PROGRAM Axis_06_Function_Blocks
VAR
END_VAR

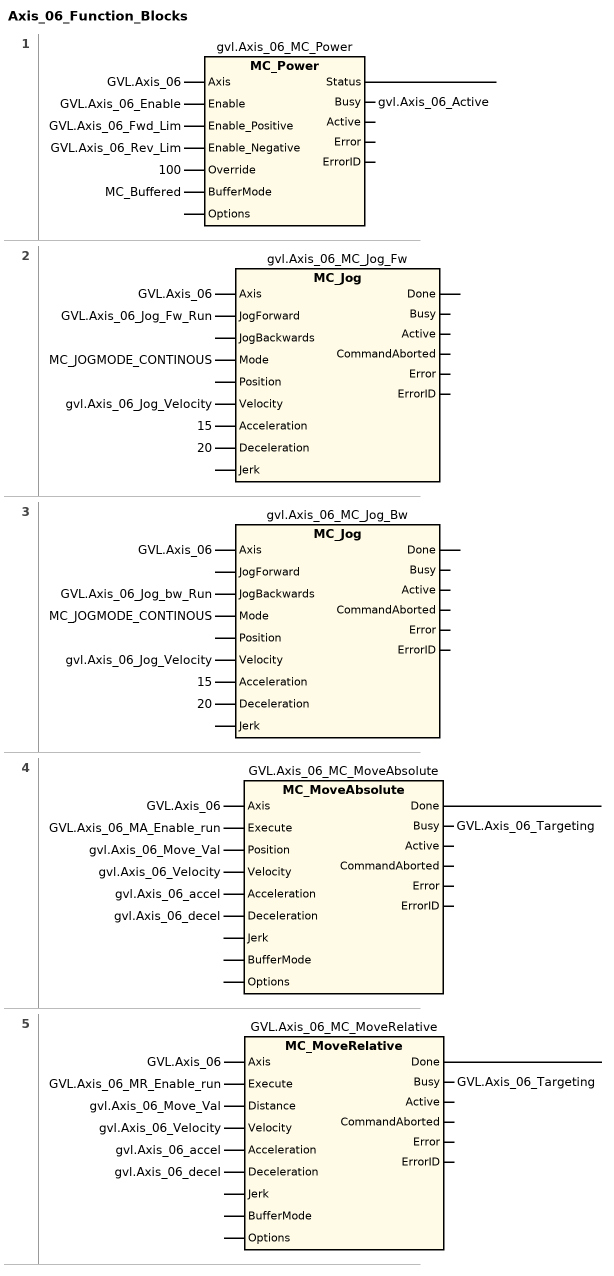
// NETWORK 1
gvl.Axis_06_MC_Power(
    Axis := GVL.Axis_06,
    Enable := GVL.Axis_06_Enable,
    Enable_Positive := GVL.Axis_06_Fwd_Lim,
    Enable_Negative := GVL.Axis_06_Rev_Lim,
    Override := 100,
    BufferMode := MC_Buffered,
    Busy => gvl.Axis_06_Active); // MC_Power

// NETWORK 2
gvl.Axis_06_MC_Jog_Fw(
    Axis := GVL.Axis_06,
    JogForward := GVL.Axis_06_Jog_Fw_Run,
    Mode := MC_JOGMODE_CONTINOUS,
    Velocity := gvl.Axis_06_Jog_Velocity,
    Acceleration := 15,
    Deceleration := 20); // MC_Jog

// NETWORK 3
gvl.Axis_06_MC_Jog_Bw(
    Axis := GVL.Axis_06,
    JogBackwards := GVL.Axis_06_Jog_bw_Run,
    Mode := MC_JOGMODE_CONTINOUS,
    Velocity := gvl.Axis_06_Jog_Velocity,
    Acceleration := 15,
    Deceleration := 20); // MC_Jog

// NETWORK 4
GVL.Axis_06_MC_MoveAbsolute(
    Axis := GVL.Axis_06,
    Execute := GVL.Axis_06_MA_Enable_run,
    Position := gvl.Axis_06_Move_Val,
    Velocity := gvl.Axis_06_Velocity,
    Acceleration := gvl.Axis_06_accel,
    Deceleration := gvl.Axis_06_decel,
    Busy => GVL.Axis_06_Targeting); // MC_MoveAbsolute

// NETWORK 5
GVL.Axis_06_MC_MoveRelative(
    Axis := GVL.Axis_06,
    Execute := GVL.Axis_06_MR_Enable_run,
    Distance := gvl.Axis_06_Move_Val,
    Velocity := gvl.Axis_06_Velocity,
    Acceleration := gvl.Axis_06_accel,
    Deceleration := gvl.Axis_06_decel,
    Busy => GVL.Axis_06_Targeting); // MC_MoveRelative

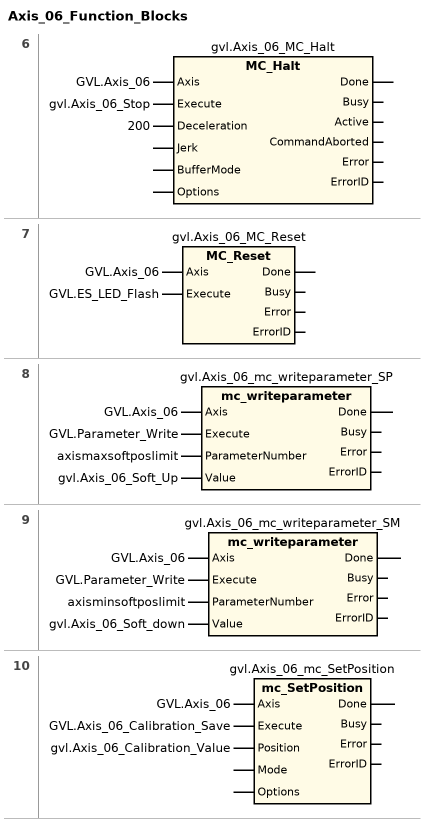
// NETWORK 6
gvl.Axis_06_MC_Halt(Axis := GVL.Axis_06, Execute := gvl.Axis_06_Stop, Deceleration := 200); // MC_Halt

// NETWORK 7
gvl.Axis_06_MC_Reset(Axis := GVL.Axis_06, Execute := GVL.ES_LED_Flash); // MC_Reset

// NETWORK 8
gvl.Axis_06_mc_writeparameter_SP(
    Axis := GVL.Axis_06,
    Execute := GVL.Parameter_Write,
    ParameterNumber := axismaxsoftposlimit,
    Value := gvl.Axis_06_Soft_Up); // mc_writeparameter

// NETWORK 9
gvl.Axis_06_mc_writeparameter_SM(
    Axis := GVL.Axis_06,
    Execute := GVL.Parameter_Write,
    ParameterNumber := axisminsoftposlimit,
    Value := gvl.Axis_06_Soft_down); // mc_writeparameter

// NETWORK 10
gvl.Axis_06_mc_SetPosition(
    Axis := GVL.Axis_06,
    Execute := GVL.Axis_06_Calibration_Save,
    Position := gvl.Axis_06_Calibration_Value); // mc_SetPosition

END_PROGRAM

(* stored: Version 1.1.0.1, ProductVersion 3.1.4022.12
   POU Axis_06_Function_Blocks: Id {6837440c-f64d-43c4-9383-6dac06a76fe4}, SpecialFunc None *)
